Fanuc KAREL source: KCL_NO_WAIT.kl

PROGRAM T
%NOLOCKGROUP
VAR
 v0 : STRING[40]
 v1 : INTEGER
BEGIN
 KCL_NO_WAIT(v0, v1)
END T
